// TwinCAT 3 PLC project SVLS_MOT
// ProgramVersion: 3.1.4026.15
// libraries:
//   LCLS General, * (SLAC)
//   lcls-twincat-math, * (SLAC - LCLS)
//   lcls-twincat-motion, * (SLAC)
//   PMPS, * (SLAC - LCLS)
//   Tc2_MC2, * (Beckhoff Automation GmbH)
//   Tc2_Standard, * (Beckhoff Automation GmbH)
//   Tc2_System, * (Beckhoff Automation GmbH)
//   Tc2_Utilities, * (Beckhoff Automation GmbH)
//   Tc3_Module, * (Beckhoff Automation GmbH)
//   TcUnit, * (www.tcunit.org)
// project tree:
//   DUTs/ ST_EPSLimits.TcDUT (not stored)
//   GVLs/ Main.TcGVL
//   ITFs/ I_ExternalSetpointGenerator.TcIO, I_HController.TcIO, I_CalculateHFromAngle.TcIO, I_MotionAxis.TcIO
//   / PlcTask.TcTTO, ProductionPlcTask.TcTTO, TestPlcTask.TcTTO
//   POUs/EPS/ FB_CheckEPS.TcPOU (not stored), FB_RestTimer.TcPOU (not stored), F_InRange.TcPOU (not stored), PRG_DET_Z_EPS.TcPOU
//   POUs/FBs/ FB_ExternalSetpointGenerator.TcPOU, FB_HController.TcPOU, FB_CalculateHFromAngle.TcPOU, FB_MotionAxisNC.TcPOU
//   POUs/ PRG_Main.TcPOU
//   Test/ FB_CalculateHFromAngle_Test.TcPOU, FB_HController_Test.TcPOU, FB_ExternalSetpointGenerator_Test.TcPOU, PRG_Test.TcPOU
// real-time tasks:
//   TASK PlcTask: cycle T#10ms, priority 20, ADS port 350
//   TASK TestPlcTask: cycle T#10ms, priority 1, ADS port 351
//   TASK ProductionPlcTask: cycle T#10ms, priority 2, ADS port 352
// motion (NC):
//   TASK SVLS_MOTION SAF: cycle T#2ms, priority 4, ADS port 501
//   TASK SVLS_MOTION SVB: cycle T#10ms, priority 8, ADS port 511
//   AXIS ExternalSetpointGenerator_Test2 (id 10)
//     OtherSettings: AllowMotionCmdToSlave=true, AllowMotionCmdToExtSetGenAxis=true
//     encoder EncType=1
//     drive DrvType=5
//       Analog: TorqueSetpointScale=10, ScaleFactorActTorque=0.1
//       TimeComp: TaskDelayCycles=1
//     controller CtrType=1
//       CtrPara: PriorControlFactor=1
//         Observer: BandWidth=20
//   AXIS ExternalSetpointGenerator_Test1 (id 9)
//     OtherSettings: AllowMotionCmdToSlave=true, AllowMotionCmdToExtSetGenAxis=true
//     encoder EncType=1
//     drive DrvType=5
//       Analog: TorqueSetpointScale=10, ScaleFactorActTorque=0.1
//       TimeComp: TaskDelayCycles=1
//     controller CtrType=1
//       CtrPara: PriorControlFactor=1
//         Observer: BandWidth=20
//   AXIS HControllerDetAngle_Test1 (id 11)
//     OtherSettings: AllowMotionCmdToSlave=true
//     encoder EncType=1
//     drive DrvType=5
//       Analog: TorqueSetpointScale=10, ScaleFactorActTorque=0.1
//       TimeComp: TaskDelayCycles=1
//     controller CtrType=1
//       CtrPara: PriorControlFactor=1
//         Observer: BandWidth=20
//   AXIS HControllerDetH_Test1 (id 12)
//     OtherSettings: AllowMotionCmdToSlave=true, AllowMotionCmdToExtSetGenAxis=true
//     encoder EncType=29
//       EncPara: ScaleFactorNumerator=1e-06, MaxCount=#xffffffff, MaxCountHighDWord=#x0000001f
//     drive DrvType=5
//       Analog: TorqueSetpointScale=10, ScaleFactorActTorque=0.1
//       TimeComp: TaskDelayCycles=1
//     controller CtrType=1
//       CtrPara: PriorControlFactor=1
//         PosDiffControl: Enable=false
//         Observer: BandWidth=20
//   AXIS M1_DET_Y_Angle (id 1)
//     General: UnitName=Degree
//     Dynamic: AccelerationMaximum=0.572958, DecelerationMaximum=0.572958, Acceleration=0.57, Deceleration=0.57
//     Velo: Maximum=0.02
//     OtherSettings: AllowMotionCmdToSlave=true
//     encoder EncType=29
//       EncPara: ScaleFactorNumerator=8.3819032e-08, Offset=-11223.9805, MaxCount=#xffffffff, MaxCountHighDWord=#x0000001f, ReferenceSystem=1
//         FilterTime: TVelo=0.1
//         Inc: RefSoftSyncMask=#x0000ffff
//     drive DrvType=24
//       Analog: VeloReferenz=0.025492, TorqueSetpointScale=10, ScaleFactorActTorque=0.1
//       TimeComp: TaskDelayCycles=1
//     controller CtrType=1
//       CtrPara: PriorControlFactor=1
//         PosDiffControl: Enable=false, Range=0.06
//         Observer: BandWidth=20
//   AXIS M2_DET_Z (id 2)
//     Dynamic: AccelerationMaximum=50, DecelerationMaximum=50, Acceleration=50, Deceleration=50
//     Velo: RefSearch=0.1, RefSync=0.1, SlowManual=0.25, FastManual=0.5, Maximum=0.5
//     TargetPosControl: Range=0.01
//     OtherSettings: AllowMotionCmdToSlave=true
//     encoder EncType=29
//       EncPara: ScaleFactorNumerator=5e-05, Offset=-6871872.3264, MaxCount=#xffffffff, MaxCountHighDWord=#x0000001f
//         SoftEndMinControl: Enable=true, Range=-53.8
//         SoftEndMaxControl: Enable=true, Range=51.3
//         Inc: RefSoftSyncMask=#x0000ffff
//     drive DrvType=24
//       Analog: VeloReferenz=0.5, TorqueSetpointScale=10, ScaleFactorActTorque=0.1
//       TimeComp: TaskDelayCycles=1
//     controller CtrType=1
//       CtrPara: PriorControlFactor=1
//         PosDiffControl: Range=0.07
//         Observer: BandWidth=20
//   AXIS M3_GRA_Y (id 3)
//     Dynamic: AccelerationMaximum=5, DecelerationMaximum=5, Acceleration=5, Deceleration=5, Jerk=5
//     Velo: RefSearch=0.01, RefSync=0.01, SlowManual=0.0025, FastManual=0.005, Maximum=0.05
//     PositionAreaControl: Range=0.003
//     TargetPosControl: Range=0.0002
//     OtherSettings: AllowMotionCmdToSlave=true
//     encoder EncType=29
//       EncPara: ScaleFactorNumerator=5e-05, Offset=-17.0296, MaxCount=#xffffffff, MaxCountHighDWord=#x0000001f
//         SoftEndMinControl: Enable=true, Range=-1.11
//         SoftEndMaxControl: Enable=true, Range=1.35
//         Inc: RefSoftSyncMask=#x0000ffff
//     drive DrvType=24
//       DrvPara: Inverse=true
//         Analog: VeloReferenz=0.106, TorqueSetpointScale=10, ScaleFactorActTorque=0.1
//         TimeComp: TaskDelayCycles=1
//     controller CtrType=1
//       CtrPara: PriorControlFactor=1
//         PosDiffControl: Range=0.1
//         Observer: BandWidth=20
//   AXIS M8_Det_Y_H (id 8)
//     Dynamic: AccelerationMaximum=100, DecelerationMaximum=100, Acceleration=1, Deceleration=1, Jerk=10
//     Velo: RefSearch=0.1, RefSync=0.1, SlowManual=0.25, FastManual=0.45, Maximum=0.25
//     PositionAreaControl: Enable=false, Range=1
//     TargetPosControl: Range=1, Time=1
//     OtherSettings: AllowMotionCmdToSlave=true, AllowMotionCmdToExtSetGenAxis=true, PulseDistancePos=1, PulseDistanceNeg=1
//     encoder EncType=29
//       EncPara: ScaleFactorNumerator=1e-06, MaxCount=#xffffffff, MaxCountHighDWord=#x0000001f
//         FilterTime: TVelo=1
//         SoftEndMinControl: Enable=true, Range=113
//         SoftEndMaxControl: Enable=true, Range=256
//         Inc: RefSoftSyncMask=#x0000ffff
//     drive DrvType=24
//       Analog: VeloReferenz=0.5, TorqueSetpointScale=10, ScaleFactorActTorque=0.1
//       TimeComp: TaskDelayCycles=1
//     controller CtrType=1
//       CtrPara: PriorControlFactor=1
//         PosDiffControl: Enable=false, Range=0.1
//         PID: PosKp=0
//         Observer: BandWidth=20
// I/O:
//   DEVICE Device 1 (EtherCAT), AmsNetId 199.4.42.250.2.1
//     EK1200_01_00 [EK1200-5000 EtherCAT Power supply (2A E-Bus)]
//       EL6070_01_00 [EL6070 1Ch. Licensing-Terminal]
//       EL7047_01_01-DET_Y [EL7047 1Ch. Stepper motor output stage (50V, 5A)]
//       EL5042_01_02-DET_Y-DET_Z [EL5042 2Ch. BiSS-C Encoder]
//       EL7047_01_03-DET_Z [EL7047 1Ch. Stepper motor output stage (50V, 5A)]
//       EL7047_01_04-GRT_Y [EL7047 1Ch. Stepper motor output stage (50V, 5A)]
//       EL5042_01_05-GRT_Y-SP5 [EL5042 2Ch. BiSS-C Encoder]
//       EL5042_01_06-SP1-SP2 [EL5042 2Ch. BiSS-C Encoder]
//       EL5042_01_07-SP3-SP4 [EL5042 2Ch. BiSS-C Encoder]
//       EL9011_01_Endstop [EL9011 End Terminal]
// variable links:
//   (this object) <-> Device 1 (EtherCAT)/EK1200_01_00/EL5042_01_02-DET_Y-DET_Z
//     Enc/Inputs/In/nComState @bit 1 <-> WcState/InputToggle
//     Enc/Inputs/In/nComState <-> WcState/WcState
//     Enc/Inputs/In/nDataIn1 <-> FB Inputs Channel 1/Position
//     Enc/Inputs/In/nDataIn1 <-> FB Inputs Channel 2/Position
//     Enc/Inputs/In/nState1 @bit 12 <-> FB Inputs Channel 1/Status/Diag
//     Enc/Inputs/In/nState1 @bit 12 <-> FB Inputs Channel 2/Status/Diag
//     Enc/Inputs/In/nState1 @bit 1 <-> FB Inputs Channel 1/Status/Error
//     Enc/Inputs/In/nState1 @bit 1 <-> FB Inputs Channel 2/Status/Error
//     Enc/Inputs/In/nState1 @bit 14 <-> FB Inputs Channel 1/Status/Input cycle counter
//     Enc/Inputs/In/nState1 @bit 14 <-> FB Inputs Channel 2/Status/Input cycle counter
//     Enc/Inputs/In/nState1 @bit 2 <-> FB Inputs Channel 1/Status/Ready
//     Enc/Inputs/In/nState1 @bit 2 <-> FB Inputs Channel 2/Status/Ready
//     Enc/Inputs/In/nState1 @bit 13 <-> FB Inputs Channel 1/Status/TxPDO State
//     Enc/Inputs/In/nState1 @bit 13 <-> FB Inputs Channel 2/Status/TxPDO State
//     Enc/Inputs/In/nState1 <-> FB Inputs Channel 1/Status/Warning
//     Enc/Inputs/In/nState1 <-> FB Inputs Channel 2/Status/Warning
//   (this object) <-> Device 1 (EtherCAT)/EK1200_01_00/EL7047_01_01-DET_Y
//     Drive/Inputs/In/nState1 @bit 3 <-> STM Status/Status/Error
//     Drive/Inputs/In/nState1 @bit 7 <-> STM Status/Status/Motor stall
//     Drive/Inputs/In/nState1 @bit 5 <-> STM Status/Status/Moving negative
//     Drive/Inputs/In/nState1 @bit 4 <-> STM Status/Status/Moving positive
//     Drive/Inputs/In/nState1 @bit 1 <-> STM Status/Status/Ready
//     Drive/Inputs/In/nState1 <-> STM Status/Status/Ready to enable
//     Drive/Inputs/In/nState1 @bit 6 <-> STM Status/Status/Torque reduced
//     Drive/Inputs/In/nState1 @bit 2 <-> STM Status/Status/Warning
//     Drive/Inputs/In/nState2 @bit 3 <-> STM Status/Status/Digital input 1
//     Drive/Inputs/In/nState2 @bit 4 <-> STM Status/Status/Digital input 2
//     Drive/Inputs/In/nState2 @bit 5 <-> STM Status/Status/Sync error
//     Drive/Inputs/In/nState2 @bit 7 <-> STM Status/Status/TxPDO Toggle
//     Drive/Inputs/In/nState4 @bit 1 <-> WcState/InputToggle
//     Drive/Inputs/In/nState4 <-> WcState/WcState
//     Drive/Outputs/Out/nCtrl1 <-> STM Control/Control/Enable
//     Drive/Outputs/Out/nCtrl1 @bit 2 <-> STM Control/Control/Reduce torque
//     Drive/Outputs/Out/nCtrl1 @bit 1 <-> STM Control/Control/Reset
//     Drive/Outputs/Out/nCtrl2 @bit 3 <-> STM Control/Control/Digital output 1
//     Drive/Outputs/Out/nDataOut2[0] <-> STM Velocity/Velocity
//   (this object) <-> Device 1 (EtherCAT)/EK1200_01_00/EL7047_01_03-DET_Z
//     Drive/Inputs/In/nState1 @bit 3 <-> STM Status/Status/Error
//     Drive/Inputs/In/nState1 @bit 7 <-> STM Status/Status/Motor stall
//     Drive/Inputs/In/nState1 @bit 5 <-> STM Status/Status/Moving negative
//     Drive/Inputs/In/nState1 @bit 4 <-> STM Status/Status/Moving positive
//     Drive/Inputs/In/nState1 @bit 1 <-> STM Status/Status/Ready
//     Drive/Inputs/In/nState1 <-> STM Status/Status/Ready to enable
//     Drive/Inputs/In/nState1 @bit 6 <-> STM Status/Status/Torque reduced
//     Drive/Inputs/In/nState1 @bit 2 <-> STM Status/Status/Warning
//     Drive/Inputs/In/nState2 @bit 3 <-> STM Status/Status/Digital input 1
//     Drive/Inputs/In/nState2 @bit 4 <-> STM Status/Status/Digital input 2
//     Drive/Inputs/In/nState2 @bit 5 <-> STM Status/Status/Sync error
//     Drive/Inputs/In/nState2 @bit 7 <-> STM Status/Status/TxPDO Toggle
//     Drive/Inputs/In/nState4 @bit 1 <-> WcState/InputToggle
//     Drive/Inputs/In/nState4 <-> WcState/WcState
//     Drive/Outputs/Out/nCtrl1 <-> STM Control/Control/Enable
//     Drive/Outputs/Out/nCtrl1 @bit 2 <-> STM Control/Control/Reduce torque
//     Drive/Outputs/Out/nCtrl1 @bit 1 <-> STM Control/Control/Reset
//     Drive/Outputs/Out/nCtrl2 @bit 3 <-> STM Control/Control/Digital output 1
//     Drive/Outputs/Out/nDataOut2[0] <-> STM Velocity/Velocity
//   (this object) <-> Device 1 (EtherCAT)/EK1200_01_00/EL5042_01_05-GRT_Y-SP5
//     Enc/Inputs/In/nComState @bit 1 <-> WcState/InputToggle
//     Enc/Inputs/In/nComState <-> WcState/WcState
//     Enc/Inputs/In/nDataIn1 <-> FB Inputs Channel 1/Position
//     Enc/Inputs/In/nState1 @bit 12 <-> FB Inputs Channel 1/Status/Diag
//     Enc/Inputs/In/nState1 @bit 1 <-> FB Inputs Channel 1/Status/Error
//     Enc/Inputs/In/nState1 @bit 14 <-> FB Inputs Channel 1/Status/Input cycle counter
//     Enc/Inputs/In/nState1 @bit 2 <-> FB Inputs Channel 1/Status/Ready
//     Enc/Inputs/In/nState1 @bit 13 <-> FB Inputs Channel 1/Status/TxPDO State
//     Enc/Inputs/In/nState1 <-> FB Inputs Channel 1/Status/Warning
//   (this object) <-> Device 1 (EtherCAT)/EK1200_01_00/EL7047_01_04-GRT_Y
//     Drive/Inputs/In/nState1 @bit 3 <-> STM Status/Status/Error
//     Drive/Inputs/In/nState1 @bit 7 <-> STM Status/Status/Motor stall
//     Drive/Inputs/In/nState1 @bit 5 <-> STM Status/Status/Moving negative
//     Drive/Inputs/In/nState1 @bit 4 <-> STM Status/Status/Moving positive
//     Drive/Inputs/In/nState1 @bit 1 <-> STM Status/Status/Ready
//     Drive/Inputs/In/nState1 <-> STM Status/Status/Ready to enable
//     Drive/Inputs/In/nState1 @bit 6 <-> STM Status/Status/Torque reduced
//     Drive/Inputs/In/nState1 @bit 2 <-> STM Status/Status/Warning
//     Drive/Inputs/In/nState2 @bit 3 <-> STM Status/Status/Digital input 1
//     Drive/Inputs/In/nState2 @bit 4 <-> STM Status/Status/Digital input 2
//     Drive/Inputs/In/nState2 @bit 5 <-> STM Status/Status/Sync error
//     Drive/Inputs/In/nState2 @bit 7 <-> STM Status/Status/TxPDO Toggle
//     Drive/Inputs/In/nState4 @bit 1 <-> WcState/InputToggle
//     Drive/Inputs/In/nState4 <-> WcState/WcState
//     Drive/Outputs/Out/nCtrl1 <-> STM Control/Control/Enable
//     Drive/Outputs/Out/nCtrl1 @bit 2 <-> STM Control/Control/Reduce torque
//     Drive/Outputs/Out/nCtrl1 @bit 1 <-> STM Control/Control/Reset
//     Drive/Outputs/Out/nCtrl2 @bit 3 <-> STM Control/Control/Digital output 1
//     Drive/Outputs/Out/nDataOut2[0] <-> STM Velocity/Velocity
//   SVLS_MOT Instance <-> Device 1 (EtherCAT)/EK1200_01_00/EL5042_01_02-DET_Y-DET_Z
//     ProductionPlcTask Inputs/Main.M1.nRawEncoderULINT <-> FB Inputs Channel 1/Position
//     ProductionPlcTask Inputs/Main.M2.nRawEncoderULINT <-> FB Inputs Channel 2/Position
//   SVLS_MOT Instance <-> Device 1 (EtherCAT)/EK1200_01_00/EL5042_01_05-GRT_Y-SP5
//     ProductionPlcTask Inputs/Main.M3.nRawEncoderULINT <-> FB Inputs Channel 1/Position
//   SVLS_MOT Instance <-> Device 1 (EtherCAT)/EK1200_01_00/EL7047_01_01-DET_Y
//     ProductionPlcTask Inputs/Main.M1.bLimitBackwardEnable <-> STM Status/Status/Digital input 2
//     ProductionPlcTask Inputs/Main.M8.bLimitBackwardEnable <-> STM Status/Status/Digital input 2
//     ProductionPlcTask Inputs/Main.M1.bLimitForwardEnable <-> STM Status/Status/Digital input 1
//     ProductionPlcTask Inputs/Main.M8.bLimitForwardEnable <-> STM Status/Status/Digital input 1
//   SVLS_MOT Instance <-> Device 1 (EtherCAT)/EK1200_01_00/EL7047_01_03-DET_Z
//     ProductionPlcTask Inputs/Main.M2.bLimitBackwardEnable <-> STM Status/Status/Digital input 2
//     ProductionPlcTask Inputs/Main.M2.bLimitForwardEnable <-> STM Status/Status/Digital input 1
//   SVLS_MOT Instance <-> Device 1 (EtherCAT)/EK1200_01_00/EL7047_01_04-GRT_Y
//     ProductionPlcTask Inputs/Main.M3.bLimitBackwardEnable <-> STM Status/Status/Digital input 2
//     ProductionPlcTask Inputs/Main.M3.bLimitForwardEnable <-> STM Status/Status/Digital input 1
//   SVLS_MOT Instance <-> SVLS_MOTION SAF/Axes/ExternalSetpointGenerator_Test1
//     TestPlcTask Inputs/PRG_Test.AxisReference_ExternalSetpointGenerator_Test1.NcToPlc <-> Outputs/ToPlc
//     TestPlcTask Outputs/PRG_Test.AxisReference_ExternalSetpointGenerator_Test1.PlcToNc <-> Inputs/FromPlc
//   SVLS_MOT Instance <-> SVLS_MOTION SAF/Axes/ExternalSetpointGenerator_Test2
//     TestPlcTask Inputs/PRG_Test.AxisReference_ExternalSetpointGenerator_Test2.NcToPlc <-> Outputs/ToPlc
//     TestPlcTask Outputs/PRG_Test.AxisReference_ExternalSetpointGenerator_Test2.PlcToNc <-> Inputs/FromPlc
//   SVLS_MOT Instance <-> SVLS_MOTION SAF/Axes/HControllerDetAngle_Test1
//     TestPlcTask Inputs/PRG_Test.stMotionStage_HControllerDetAngle_Test1.Axis.NcToPlc <-> Outputs/ToPlc
//     TestPlcTask Outputs/PRG_Test.stMotionStage_HControllerDetAngle_Test1.Axis.PlcToNc <-> Inputs/FromPlc
//   SVLS_MOT Instance <-> SVLS_MOTION SAF/Axes/HControllerDetH_Test1
//     PlcTask Outputs/PRG_Test.fbHController_Test.nDetAngleEncoderComState_Test1 <-> Enc/Inputs/In/nComState
//     PlcTask Outputs/PRG_Test.fbHController_Test.nDetAngleEncoderState1_Test1 <-> Enc/Inputs/In/nState1
//     TestPlcTask Inputs/PRG_Test.stMotionStage_HControllerDetH_Test1.Axis.NcToPlc <-> Outputs/ToPlc
//     TestPlcTask Outputs/PRG_Test.stMotionStage_HControllerDetH_Test1.Axis.PlcToNc <-> Inputs/FromPlc
//   SVLS_MOT Instance <-> SVLS_MOTION SAF/Axes/M1_DET_Y_Angle
//     ProductionPlcTask Inputs/Main.M1.Axis.NcToPlc <-> Outputs/ToPlc
//     ProductionPlcTask Outputs/Main.M1.Axis.PlcToNc <-> Inputs/FromPlc
//   SVLS_MOT Instance <-> SVLS_MOTION SAF/Axes/M2_DET_Z
//     ProductionPlcTask Inputs/Main.M2.Axis.NcToPlc <-> Outputs/ToPlc
//     ProductionPlcTask Outputs/Main.M2.Axis.PlcToNc <-> Inputs/FromPlc
//   SVLS_MOT Instance <-> SVLS_MOTION SAF/Axes/M3_GRA_Y
//     ProductionPlcTask Inputs/Main.M3.Axis.NcToPlc <-> Outputs/ToPlc
//     ProductionPlcTask Outputs/Main.M3.Axis.PlcToNc <-> Inputs/FromPlc
//   SVLS_MOT Instance <-> SVLS_MOTION SAF/Axes/M8_Det_Y_H
//     ProductionPlcTask Inputs/Main.M8.Axis.NcToPlc <-> Outputs/ToPlc
//     ProductionPlcTask Outputs/Main.M8.Axis.PlcToNc <-> Inputs/FromPlc
//     ProductionPlcTask Outputs/PRG_Main.fbHController.nEncoderCounts <-> Enc/Inputs/In/nDataIn1
//   SVLS_MOT Instance <-> SVLS_MOT/SVLS_MOT Instance
//     ProductionPlcTask Inputs/Main.M8.nRawEncoderULINT <-> ProductionPlcTask Outputs/PRG_Main.fbHController.nEncoderCounts
//     ProductionPlcTask Outputs/PRG_Main.fbHController.nEncoderCounts <-> ProductionPlcTask Inputs/Main.M8.nRawEncoderULINT

CONFIGURATION SVLS_MOT
    RESOURCE PLC ON TwinCAT3
        TASK PlcTask(INTERVAL := T#10ms, PRIORITY := 20);
        TASK ProductionPlcTask(INTERVAL := T#10ms, PRIORITY := 2);
        TASK TestPlcTask(INTERVAL := T#10ms, PRIORITY := 1);
        PROGRAM PRG_Main WITH ProductionPlcTask : PRG_Main;
        PROGRAM PRG_Test WITH TestPlcTask : PRG_Test;
    END_RESOURCE
END_CONFIGURATION

// ---- GVLs/Main.TcGVL

{attribute 'qualified_only'}
VAR_GLOBAL
    {attribute 'pytmc' := 'pv: CRIXS:SVLS:DET:MMS:Y_Angle'}
    {attribute 'TcLinkTo' := '.bLimitForwardEnable  := TIIB[EL7047_01_01-DET_Y]^STM Status^Status^Digital input 1;
                              .bLimitBackwardEnable := TIIB[EL7047_01_01-DET_Y]^STM Status^Status^Digital input 2;
                              .nRawEncoderULINT     := TIIB[EL5042_01_02-DET_Y-DET_Z]^FB Inputs Channel 1^Position'}
    M1: ST_MotionStage := (sName := 'CRIXS:SVLS:DET:MMS:Y_Angle');

    {attribute 'pytmc' := 'pv: CRIXS:SVLS:DET:MMS:Z'}
    {attribute 'TcLinkTo' := '.bLimitForwardEnable  := TIIB[EL7047_01_03-DET_Z]^STM Status^Status^Digital input 1;
                              .bLimitBackwardEnable := TIIB[EL7047_01_03-DET_Z]^STM Status^Status^Digital input 2;
                              .nRawEncoderULINT     := TIIB[EL5042_01_02-DET_Y-DET_Z]^FB Inputs Channel 2^Position'}
    M2: ST_MotionStage := (sName := 'CRIXS:SVLS:DET:MMS:Z');

    {attribute 'pytmc' := 'pv: CRIXS:SVLS:GRA:MMS:Y'}
    {attribute 'TcLinkTo' := '.bLimitForwardEnable  := TIIB[EL7047_01_04-GRT_Y]^STM Status^Status^Digital input 1;
                              .bLimitBackwardEnable := TIIB[EL7047_01_04-GRT_Y]^STM Status^Status^Digital input 2;
                              .nRawEncoderULINT     := TIIB[EL5042_01_05-GRT_Y-SP5]^FB Inputs Channel 1^Position'}
    M3: ST_MotionStage := (sName := 'CRIXS:SVLS:GRA:MMS:Y');

    {attribute 'pytmc' := 'pv:	CRIXS:SVLS:DET:MMS:Y_H'}
    {attribute 'TcLinkTo' := '.bLimitForwardEnable  := TIIB[EL7047_01_01-DET_Y]^STM Status^Status^Digital input 1;
                              .bLimitBackwardEnable := TIIB[EL7047_01_01-DET_Y]^STM Status^Status^Digital input 2;
                              .nRawEncoderULINT     := TIPC^SVLS_MOT^SVLS_MOT Instance^ProductionPlcTask Outputs^PRG_Main.fbHController.nEncoderCounts'}
    M8 : ST_MotionStage := (sName := 'CRIXS:SVLS:DET:MMS:Y_H');
	
END_VAR

// ---- ITFs/I_ExternalSetpointGenerator.TcIO
INTERFACE I_ExternalSetpointGenerator


METHOD Disable
VAR_OUTPUT
    Done : BOOL;
    Busy : BOOL;
    Error : BOOL;
    ErrorID : UDINT;
    Enabled : BOOL;
END_VAR
END_METHOD

PROPERTY DisableBusy : BOOL
GET
END_GET
END_PROPERTY

PROPERTY DisableDone : BOOL
GET
END_GET
END_PROPERTY


METHOD Enable
VAR_OUTPUT
    Done : BOOL;
    Busy : BOOL;
    Error : BOOL;
    ErrorID : UDINT;
    Enabled : BOOL;
END_VAR
END_METHOD

PROPERTY EnableBusy : BOOL
GET
END_GET
END_PROPERTY

PROPERTY EnableDone : BOOL
GET
END_GET
END_PROPERTY

PROPERTY EnableError : BOOL
GET
END_GET
END_PROPERTY


METHOD Halt
VAR_OUTPUT
    Done : BOOL;
    Busy : BOOL;
    Active : BOOL;
    CommandAborted : BOOL;
    Error : BOOL;
    ErrorID : UDINT;
END_VAR
END_METHOD

PROPERTY HaltBusy : BOOL
GET
END_GET
END_PROPERTY

PROPERTY HaltDone : BOOL
GET
END_GET
END_PROPERTY


METHOD IsEnabled : BOOL
END_METHOD


METHOD SetAcceleraSetpoint
VAR_INPUT
    Setpoint : LREAL;
END_VAR
VAR_OUTPUT
	Error : BOOL;
	ErrorMsg : T_MaxString;
END_VAR
END_METHOD


METHOD SetPositionSetpoint
VAR_INPUT
    Setpoint : LREAL;
END_VAR
VAR_OUTPUT
	Error : BOOL;
	ErrorMsg : T_MaxString;
END_VAR
END_METHOD


METHOD SetSetpoints
VAR_INPUT
    PositionSetpoint : LREAL;
    VelocitySetpoint : LREAL;
    AcceleraSetpoint : LREAL;
END_VAR
VAR_OUTPUT
	Error : BOOL;
	ErrorMsg : T_MaxString;
END_VAR
END_METHOD


METHOD SetVelocitySetpoint
VAR_INPUT
    Setpoint : LREAL;
END_VAR
VAR_OUTPUT
	Error : BOOL;
	ErrorMsg : T_MaxString;
END_VAR
END_METHOD

END_INTERFACE

// ---- ITFs/I_HController.TcIO
INTERFACE I_HController

END_INTERFACE

// ---- ITFs/I_CalculateHFromAngle.TcIO
INTERFACE I_CalculateHFromAngle


METHOD CalculateH : LREAL
VAR_INPUT
    Radians : LREAL;
END_VAR
VAR_OUTPUT
    Error : BOOL;
    ErrorMsg : T_MaxString;
END_VAR
END_METHOD


METHOD CalculateHVelocity : LREAL
VAR_INPUT
    Radians : LREAL;
    RadiansPerSecond : LREAL;
END_VAR
VAR_OUTPUT
    Error : BOOL;
    ErrorMsg : T_MaxString;
END_VAR
END_METHOD

END_INTERFACE

// ---- ITFs/I_MotionAxis.TcIO

INTERFACE I_MotionAxis


METHOD GetAxisRef : REFERENCE TO AXIS_REF
END_METHOD


METHOD GetPowerOverride : LREAL
END_METHOD

PROPERTY MeasuredAcceleration : LREAL
GET
END_GET
END_PROPERTY

PROPERTY MeasuredPosition : LREAL
GET
END_GET
END_PROPERTY

PROPERTY MeasuredVelocity : LREAL
GET
END_GET
END_PROPERTY


METHOD MoveAbsolute
VAR_INPUT
    Position : LREAL; 
    Velocity : LREAL; 
    Acceleration : LREAL := 0.0; 
    Deceleration : LREAL := 0.0; 
    Jerk : LREAL := 0.0;
    BufferMode : MC_BufferMode := MC_BufferMode.MC_Aborting;
END_VAR
VAR_OUTPUT
    Done : BOOL;
    Busy : BOOL;
    Active : BOOL;
    CommandAborted : BOOL;
    Error : BOOL;
    ErrorID : UDINT;
    ErrorStr : T_MaxString;
END_VAR
END_METHOD

PROPERTY MoveAbsoluteBusy : BOOL
GET
END_GET
END_PROPERTY

PROPERTY MoveAbsoluteDone : BOOL
GET
END_GET
END_PROPERTY

PROPERTY MoveAbsoluteError : BOOL
GET
END_GET
END_PROPERTY

PROPERTY MoveAbsoluteErrorID : UDINT
GET
END_GET
END_PROPERTY

PROPERTY MoveAbsoluteTargetAcceleration : LREAL
GET
END_GET
END_PROPERTY

PROPERTY MoveAbsoluteTargetDeceleration : LREAL
GET
END_GET
END_PROPERTY

PROPERTY MoveAbsoluteTargetJerk : LREAL
GET
END_GET
END_PROPERTY

PROPERTY MoveAbsoluteTargetPosition : LREAL
GET
END_GET
END_PROPERTY

PROPERTY MoveAbsoluteTargetVelocity : LREAL
GET
END_GET
END_PROPERTY

PROPERTY NegativeMotionIsEnabled : BOOL
GET
END_GET
END_PROPERTY

PROPERTY PositiveMotionIsEnabled : BOOL
GET
END_GET
END_PROPERTY


METHOD Power
VAR_INPUT
    Enable : BOOL;
    Enable_Positive : BOOL;
    Enable_Negative : BOOL;
    Override : LREAL := 100.0; (* in percent from 0 to 100 *)
    BufferMode : MC_BufferMode := MC_BufferMode.MC_Aborting;
END_VAR
VAR_OUTPUT
    Status : BOOL;
    Busy : BOOL;
    Active : BOOL;
    Error : BOOL;
    ErrorID : UDINT;
    ErrorStr : T_MaxString;
END_VAR
END_METHOD

PROPERTY PowerError : BOOL
GET
END_GET
END_PROPERTY

PROPERTY PowerErrorID : UDINT
GET
END_GET
END_PROPERTY

PROPERTY PowerIsEnabled : BOOL
GET
END_GET
END_PROPERTY

PROPERTY PowerOverride : LREAL
GET
END_GET
END_PROPERTY

PROPERTY PowerStatus : BOOL
GET
END_GET
END_PROPERTY


METHOD Reset
VAR_OUTPUT
    Done    : BOOL;
    Busy    : BOOL;
    Error   : BOOL;
    ErrorID : UDINT;
    ErrorStr : T_MaxString;
END_VAR
END_METHOD


PROPERTY SetpointAcceleration : LREAL
GET
END_GET
END_PROPERTY


PROPERTY SetpointJerk : LREAL
GET
END_GET
END_PROPERTY


PROPERTY SetpointPosition : LREAL
GET
END_GET
END_PROPERTY


PROPERTY SetpointVelocity : LREAL
GET
END_GET
END_PROPERTY


METHOD SetPowerOverride
VAR_INPUT
    Override : LREAL; (* in percent from 0 to 100 *)
END_VAR
VAR_OUTPUT
    Status : BOOL;
    Busy : BOOL;
    Active : BOOL;
    Error : BOOL;
    ErrorID : UDINT;
    ErrorStr : T_MaxString;
END_VAR
END_METHOD

END_INTERFACE

// ---- POUs/PRG_Main.TcPOU

PROGRAM PRG_Main
VAR
    fbDetYAngle : FB_MotionStage;
    fbDetZ : FB_MotionStage;
    fbGraY : FB_MotionStage;
    fbDetYH : FB_MotionStage;
    bInit : BOOL := TRUE;

    fbMotionAxisDetAngle : FB_MotionAxisNC(
        AxisReference := Main.M1.Axis
    );
    fbMotionAxisDetH : FB_MotionAxisNC(
        AxisReference := Main.M8.Axis
    );
    fbCalculateHFromAngle : FB_CalculateHFromAngle(
        D_tu := 1238.29,
        R_a := 1200.10,
        R_c := 89.78
    );
    {attribute 'TcLinkTo' := '.nEncoderCount := TINC^SVLS_MOTION SAF^Axes^M8_Det_Y_H^Enc^Inputs^In^nDataIn1'}
    fbHController : FB_HController(
        iMotionAxisDetAngle := fbMotionAxisDetAngle,
        iCalculateHFromAngle := fbCalculateHFromAngle,
        stMotionStageAxisDetAngle := Main.M1,
        stMotionStageAxisDetH := Main.M8,
        bDetHMoveAbsoluteBusy := fbDetYH.fbDriveVirtual.fbMoveAbsolute.Busy
    );
	
END_VAR


IF bInit THEN
    bInit := FALSE;

    Main.M1.bHardwareEnable := TRUE;
    Main.M1.bPowerSelf := TRUE;
    Main.M1.nBrakeMode := ENUM_StageBrakeMode.NO_BRAKE;
    Main.M1.nEnableMode := ENUM_StageEnableMode.DURING_MOTION;

    Main.M2.bHardwareEnable := TRUE;
    Main.M2.bPowerSelf := TRUE;
    Main.M2.nBrakeMode := ENUM_StageBrakeMode.NO_BRAKE;
    Main.M2.nEnableMode := ENUM_StageEnableMode.DURING_MOTION;

    Main.M3.bHardwareEnable := TRUE;
    Main.M3.bPowerSelf := TRUE;
    Main.M3.nBrakeMode := ENUM_StageBrakeMode.NO_BRAKE;
    Main.M3.nEnableMode := ENUM_StageEnableMode.DURING_MOTION;

    Main.M8.bHardwareEnable := TRUE;
    Main.M8.bPowerSelf := TRUE;
    Main.M8.nBrakeMode := ENUM_StageBrakeMode.NO_BRAKE;
    Main.M8.nEnableMode := ENUM_StageEnableMode.DURING_MOTION;
END_IF

PRG_DET_Z_EPS();

fbDetYAngle(stMotionStage:=Main.M1);
fbHController();
fbDetYH(stMotionStage:=Main.M8);
fbDetZ(stMotionStage:=Main.M2);
fbGraY(stMotionStage:=Main.M3);

END_PROGRAM

// ---- POUs/FBs/FB_MotionAxisNC.TcPOU

FUNCTION_BLOCK FB_MotionAxisNC IMPLEMENTS I_MotionAxis
VAR CONSTANT
    nOFFSET_TO_PLCTONC_AXIS_REF_CTRL : DWORD := 0;
END_VAR
VAR
    AxisReference : REFERENCE TO AXIS_REF;

    AxisReference_PLCtoNC_ControlDWord : MC.PLCTONC_AXIS_REF_CTRL;

    fbMcReset : MC_Reset;
    bCommandedReset : BOOL;

    fbMcPower : MC_Power;

    bCommandedMoveAbsolute : BOOL;
    fbMcMoveAbsolute : MC_MoveAbsolute;

    bMostRecentMoveAbsoluteDone : BOOL;
END_VAR


AxisReference.ReadStatus();

MEMCPY(
    ADR(AxisReference_PLCtoNC_ControlDWord),
    ADR(AxisReference.PlcToNc) + nOFFSET_TO_PLCTONC_AXIS_REF_CTRL,
    SIZEOF(AxisReference_PLCtoNC_ControlDWord)
);

fbMcReset(
    Axis := AxisReference,
    Execute := bCommandedReset
);
bCommandedReset := FALSE;

fbMcPower(Axis := AxisReference);

// IF bCommandedMoveAbsolute THEN
// 	ADSLOGSTR(
// 		msgCtrlMask := ADSLOG_MSGTYPE_ERROR,
// 		msgFmtStr := 'Commanded move absolute.',
// 		strArg := ''
// 	);
// END_IF

fbMcMoveAbsolute(
    Axis := AxisReference,
    Execute := bCommandedMoveAbsolute
);
bCommandedMoveAbsolute := FALSE;

IF THIS^.fbMcMoveAbsolute.Done THEN
    THIS^.bMostRecentMoveAbsoluteDone := TRUE;
END_IF

//FB_Init is always available implicitly and it is used primarily for initialization.
//The return value is not evaluated. For a specific influence, you can also declare the
//methods explicitly and provide additional code there with the standard initialization
//code. You can evaluate the return value.
METHOD FB_Init: BOOL
VAR_INPUT
    bInitRetains: BOOL; // TRUE: the retain variables are initialized (reset warm / reset cold)
    bInCopyCode: BOOL;  // TRUE: the instance will be copied to the copy code afterward (online change)

    AxisReference : REFERENCE TO AXIS_REF;
END_VAR

THIS^.AxisReference REF= AxisReference;
END_METHOD


METHOD GetAxisRef : REFERENCE TO AXIS_REF

GetAxisRef REF= THIS^.AxisReference;
END_METHOD


METHOD GetPowerOverride : LREAL

GetPowerOverride := TO_LREAL(THIS^.AxisReference.PlcToNc.Override) / 10000.0;
END_METHOD


PROPERTY MeasuredAcceleration : LREAL
GET

MeasuredAcceleration := THIS^.AxisReference.NcToPlc.ActAcc;
END_GET
END_PROPERTY


PROPERTY MeasuredPosition : LREAL
GET

MeasuredPosition := THIS^.AxisReference.NcToPlc.ActPos;
END_GET
END_PROPERTY


PROPERTY MeasuredVelocity : LREAL
GET

MeasuredVelocity := THIS^.AxisReference.NcToPlc.ActVelo;
END_GET
END_PROPERTY


METHOD MoveAbsolute
VAR_INPUT
    Position	: LREAL;
    Velocity	: LREAL;
    Acceleration	: LREAL := 0.0;
    Deceleration	: LREAL := 0.0;
    Jerk	: LREAL := 0.0;
    BufferMode	: MC_BufferMode := MC_BufferMode.MC_Aborting;
END_VAR
VAR_OUTPUT
    Done	: BOOL;
    Busy	: BOOL;
    Active	: BOOL;
    CommandAborted	: BOOL;
    Error	: BOOL;
    ErrorID	: UDINT;
    ErrorStr	: T_MaxString;
END_VAR

IF NOT MoveAbsoluteBusy THEN
    bMostRecentMoveAbsoluteDone := FALSE;

    bCommandedMoveAbsolute := TRUE;
END_IF

THIS^.fbMcMoveAbsolute(
    Axis := THIS^.AxisReference,
    Position := Position,
    Velocity := Velocity,
    Acceleration := Acceleration,
    Deceleration := Deceleration,
    Jerk := Jerk,
    BufferMode := BufferMode,
    Done => Done,
    Busy => Busy,
    Active => Active,
    CommandAborted => CommandAborted,
    Error => Error,
    ErrorID => ErrorID
);

ErrorStr := '';
END_METHOD


PROPERTY MoveAbsoluteBusy : BOOL
GET

MoveAbsoluteBusy := THIS^.fbMcMoveAbsolute.Busy;
END_GET
END_PROPERTY


PROPERTY MoveAbsoluteDone : BOOL
GET

MoveAbsoluteDone := THIS^.fbMcMoveAbsolute.Done OR THIS^.bMostRecentMoveAbsoluteDone;
END_GET
END_PROPERTY


PROPERTY MoveAbsoluteError : BOOL
GET

MoveAbsoluteError := THIS^.fbMcMoveAbsolute.Error;
END_GET
END_PROPERTY


PROPERTY MoveAbsoluteErrorID : UDINT
GET

MoveAbsoluteErrorID := THIS^.fbMcMoveAbsolute.ErrorID;
END_GET
END_PROPERTY


PROPERTY MoveAbsoluteTargetAcceleration : LREAL
GET

MoveAbsoluteTargetAcceleration := THIS^.fbMcMoveAbsolute.Acceleration;
END_GET
END_PROPERTY


PROPERTY MoveAbsoluteTargetDeceleration : LREAL
GET

MoveAbsoluteTargetDeceleration := THIS^.fbMcMoveAbsolute.Deceleration;
END_GET
END_PROPERTY


PROPERTY MoveAbsoluteTargetJerk : LREAL
GET

MoveAbsoluteTargetJerk := THIS^.fbMcMoveAbsolute.Jerk;
END_GET
END_PROPERTY


PROPERTY MoveAbsoluteTargetPosition : LREAL
GET

MoveAbsoluteTargetPosition := THIS^.fbMcMoveAbsolute.Position;
END_GET
END_PROPERTY


PROPERTY MoveAbsoluteTargetVelocity : LREAL
GET

MoveAbsoluteTargetVelocity := THIS^.fbMcMoveAbsolute.Velocity;
END_GET
END_PROPERTY


PROPERTY NegativeMotionIsEnabled : BOOL
GET

NegativeMotionIsEnabled := THIS^.AxisReference_PLCtoNC_ControlDWord.2;;
END_GET
END_PROPERTY


PROPERTY PositiveMotionIsEnabled : BOOL
GET

PositiveMotionIsEnabled := THIS^.AxisReference_PLCtoNC_ControlDWord.1;
END_GET
END_PROPERTY


METHOD Power
VAR_INPUT
    Enable	: BOOL;
    Enable_Positive	: BOOL;
    Enable_Negative	: BOOL;
    (* in percent from 0 to 100 *)
    Override	: LREAL := 100.0;
    BufferMode	: MC_BufferMode := MC_BufferMode.MC_Aborting;
END_VAR
VAR_OUTPUT
    Status	: BOOL;
    Busy	: BOOL;
    Active	: BOOL;
    Error	: BOOL;
    ErrorID	: UDINT;
    ErrorStr	: T_MaxString;
END_VAR

THIS^.fbMcPower(
    Axis := THIS^.AxisReference,
    Enable := Enable,
    Enable_Positive := Enable_Positive,
    Enable_Negative := Enable_Negative,
    Override := Override,
    BufferMode := BufferMode,
    Status => Status,
    Busy => Busy,
    Active => Active,
    Error => Error,
    ErrorID => ErrorID
);

ErrorStr := '';
END_METHOD


PROPERTY PowerError : BOOL
GET

PowerError := THIS^.fbMcPower.Error;
END_GET
END_PROPERTY


PROPERTY PowerErrorID : UDINT
GET

PowerErrorID := THIS^.fbMcPower.ErrorID;
END_GET
END_PROPERTY


METHOD PowerErrorIDToStr : T_MaxString
VAR_INPUT
    ErrorID : UDINT;
END_VAR

PowerErrorIDToStr := '';
END_METHOD


PROPERTY PowerIsEnabled : BOOL
GET

PowerIsEnabled := THIS^.AxisReference_PLCtoNC_ControlDWord.0;
END_GET
END_PROPERTY


PROPERTY PowerOverride : LREAL
GET

PowerOverride := GetPowerOverride();
END_GET
END_PROPERTY


PROPERTY PowerStatus : BOOL
GET

PowerStatus := THIS^.fbMcPower.Status;
END_GET
END_PROPERTY


METHOD Reset
VAR_OUTPUT
    Done : BOOL;
    Busy : BOOL;
    Error : BOOL;
    ErrorID : UDINT;
    ErrorStr : T_MaxString;
END_VAR

bCommandedReset := TRUE;

THIS^.fbMcReset(
    Axis := THIS^.AxisReference,
    Done => Done,
    Busy => Busy,
    Error => Error,
    ErrorID => ErrorID,
);

ErrorStr := '';
END_METHOD


PROPERTY SetpointAcceleration : LREAL
GET

SetpointAcceleration := THIS^.AxisReference.NcToPlc.SetAcc;
END_GET
END_PROPERTY


PROPERTY SetpointJerk : LREAL
GET

SetpointJerk := THIS^.AxisReference.NcToPlc.SetJerk;
END_GET
END_PROPERTY


PROPERTY SetpointPosition : LREAL
GET

SetpointPosition := THIS^.AxisReference.NcToPlc.SetPos;
END_GET
END_PROPERTY


PROPERTY SetpointVelocity : LREAL
GET

SetpointVelocity := THIS^.AxisReference.NcToPlc.SetVelo;
END_GET
END_PROPERTY


METHOD SetPowerOverride
VAR_INPUT
    (* in percent from 0 to 100 *)
    Override	: LREAL;
END_VAR
VAR_OUTPUT
    Status	: BOOL;
    Busy	: BOOL;
    Active	: BOOL;
    Error	: BOOL;
    ErrorID	: UDINT;
    ErrorStr	: T_MaxString;
END_VAR

THIS^.fbMcPower(
    Axis := THIS^.AxisReference,
    Override := Override,
    Status => Status,
    Busy => Busy,
    Error => Error,
    ErrorID => ErrorID
);

ErrorStr := '';
END_METHOD

END_FUNCTION_BLOCK

// ---- POUs/FBs/FB_CalculateHFromAngle.TcPOU

{attribute 'no_explicit_call' := 'Do not call this POU directly'}
FUNCTION_BLOCK FB_CalculateHFromAngle IMPLEMENTS I_CalculateHFromAngle
VAR
    D_tu : LREAL;
    R_c : LREAL;
    R_a : LREAL;
END_VAR


METHOD PUBLIC CalculateH : LREAL
VAR_INPUT
    Radians : LREAL;
END_VAR
VAR_OUTPUT
    Error : BOOL;
    ErrorMsg : T_MaxString;
END_VAR
VAR
    a : LREAL;
    b : LREAL;
    c : LREAL;
    d : LREAL;
    e : LREAL;
    f : LREAL;
    g : LREAL;
    h : LREAL;
    //sqrt_operand : LREAL;
END_VAR

IF R_c = 0 THEN
    Error := TRUE;
    ErrorMsg := CONCAT('R_c cannot equal 0. Value: ', TO_STRING(R_c));
    RETURN;
END_IF

a := R_a * COS(Radians);
b := D_tu - a;
c := b / R_c;

IF c < -1.0 OR c > 1.0 THEN
    Error := TRUE;
    ErrorMsg := CONCAT('Invalid angle. Value: ', TO_STRING(Radians));
    RETURN;
END_IF

d := ACOS(c);
e := SIN(d);
f := SIN(Radians);
g := R_a * f;
h := R_c * e;

CalculateH := h + g;

(*
sqrt_operand := -EXPT(R_a,2) * EXPT(COS(Angle),2) + 2 * R_a * D_tu * COS(Angle) + R_c - EXPT(D_tu,2);

IF sqrt_operand < 0.0 THEN
    Error := TRUE;
    ErrorMsg := CONCAT('Invalid angle. Value: ', TO_STRING(Angle));
    RETURN;
END_IF

CalculateH := R_a * SIN(Angle) - SQRT(sqrt_operand);
*)
END_METHOD


METHOD CalculateHVelocity : LREAL
VAR_INPUT
    Radians : LREAL;
    RadiansPerSecond : LREAL;
END_VAR
VAR_OUTPUT
    Error : BOOL;
    ErrorMsg : T_MaxString;
END_VAR
VAR
    A : LREAL;
    b : LREAL;
    b_dot : LREAL;
    C : LREAL;
    D : LREAL;
    fNumberToSqrt : LREAL;
END_VAR

A := R_a;
b := Radians;
b_dot := RadiansPerSecond;
C := R_c;
D := D_tu;
fNumberToSqrt := 1 - EXPT((D - (A * COS(b))/C), 2);

IF fNumberToSqrt <= 0 THEN
    Error := TRUE;
    ErrorMsg := 'number to sqrt was 0 or less than 0.';
    RETURN;
END_IF

CalculateHVelocity := A * b_dot * (COS(b) - (SIN(b)*(D - (COS(b))/C))/(SQRT(fNumberToSqrt)));
END_METHOD


METHOD FB_Init: BOOL
VAR_INPUT
    bInitRetains: BOOL; // TRUE: the retain variables are initialized (reset warm / reset cold)
    bInCopyCode: BOOL;  // TRUE: the instance will be copied to the copy code afterward (online change)

    D_tu : LREAL;
    R_c : LREAL;
    R_a : LREAL;
END_VAR

THIS^.D_tu := D_tu;
THIS^.R_c := R_c;
THIS^.R_a := R_a;
END_METHOD

END_FUNCTION_BLOCK

// ---- POUs/FBs/FB_HController.TcPOU

FUNCTION_BLOCK FB_HController IMPLEMENTS I_HController
VAR
    iMotionAxisDetAngle : I_MotionAxis;
    iCalculateHFromAngle : I_CalculateHFromAngle;
    stMotionStageAxisDetAngle : REFERENCE TO ST_MotionStage;
    stMotionStageAxisDetH : REFERENCE TO ST_MotionStage;
    bDetHMoveAbsoluteBusy : REFERENCE TO BOOL;

    fHPositionMeasured : LREAL;
    fHPositionSetpoint : LREAL;

    fHPositionGain : LREAL;
    fHPositionAdjustmentIntegration : LREAL;

    nEncoderCounts AT %Q* : ULINT; // nm/count

    rtMoveCmdTrigger : R_TRIG;
    ftResetTrigger : F_TRIG;
END_VAR


fHPositionMeasured := iCalculateHFromAngle.CalculateH(
    Radians := DEG_TO_RAD(iMotionAxisDetAngle.MeasuredPosition)
);

nEncoderCounts := TO_ULINT(fHPositionMeasured * 1E6);

fHPositionSetpoint := iCalculateHFromAngle.CalculateH(
    Radians := DEG_TO_RAD(iMotionAxisDetAngle.SetpointPosition)
);

rtMoveCmdTrigger(CLK := stMotionStageAxisDetAngle.bExecute);

IF rtMoveCmdTrigger.Q THEN
    stMotionStageAxisDetH.bMoveCmd := TRUE;
    stMotionStageAxisDetH.fPosition := iCalculateHFromAngle.CalculateH(
        Radians := DEG_TO_RAD(stMotionStageAxisDetAngle.fPosition)
    );
    stMotionStageAxisDetH.fVelocity := stMotionStageAxisDetH.stAxisParameters.fVeloMaximum *
        stMotionStageAxisDetAngle.fVelocity / stMotionStageAxisDetAngle.stAxisParameters.fVeloMaximum;
END_IF

ftResetTrigger(CLK := bDetHMoveAbsoluteBusy);

IF ftResetTrigger.Q THEN
    stMotionStageAxisDetAngle.bReset := TRUE;
    stMotionStageAxisDetH.bReset := TRUE;
END_IF


METHOD FB_Init: BOOL
VAR_INPUT
    bInitRetains: BOOL; // TRUE: the retain variables are initialized (reset warm / reset cold)
    bInCopyCode: BOOL;  // TRUE: the instance will be copied to the copy code afterward (online change)

    iMotionAxisDetAngle : I_MotionAxis;
    iCalculateHFromAngle : I_CalculateHFromAngle;
    stMotionStageAxisDetAngle : REFERENCE TO ST_MotionStage;
    stMotionStageAxisDetH : REFERENCE TO ST_MotionStage;
    bDetHMoveAbsoluteBusy : REFERENCE TO BOOL;

END_VAR

THIS^.iMotionAxisDetAngle := iMotionAxisDetAngle;
THIS^.iCalculateHFromAngle := iCalculateHFromAngle;
THIS^.stMotionStageAxisDetAngle REF= stMotionStageAxisDetAngle;
THIS^.stMotionStageAxisDetH REF= stMotionStageAxisDetH;
THIS^.bDetHMoveAbsoluteBusy REF= bDetHMoveAbsoluteBusy;
END_METHOD

END_FUNCTION_BLOCK

// ---- POUs/EPS/PRG_DET_Z_EPS.TcPOU
PROGRAM PRG_DET_Z_EPS
VAR
	{attribute 'pytmc' := 'pv: SVLS:DET:MMS:Z:EPS'}
    aDET_Z_EPS		: ARRAY [1 .. 2] OF ST_EPSLimits;
	
    {attribute 'pytmc' := 'pv: CRIX:DPL:MMS:X:EPS:OVRD_MODE'}
    bEPS_Override : BOOL := FALSE;
    {attribute 'pytmc' := 'pv: CRIX:DPL:MMS:X:EPS:OVRD_COUNTDOWN'}
    tEPS_TimerCountDown : STRING := TIME_TO_STRING(T#0S);
	tEPS_OVRD_RESET_TIME : TIME := T#5M;
    fbResetTimer : FB_RestTimer;
	
	
	bInit : BOOL := TRUE;
	
	fDET_Z : LREAL;
	fDET_Y_ANGLE : LREAL ;
	fDET_Y_ANGLE_VALUE : LREAL := 6;
	bYAngleBelow : BOOL;

    fbEPS : FB_EPS;
    fbCheckEPS : FB_CheckEPS;
END_VAR

fDET_Y_ANGLE := Main.M1.stAxisStatus.fActPosition;
fDET_Z := Main.M2.stAxisStatus.fActPosition;

IF bInit THEN
    // Set Inital Values
    aDET_Z_EPS[1].fBwd_Limits := -53.8;
    aDET_Z_EPS[1].fFwd_Limits := 35;
	
    aDET_Z_EPS[2].fBwd_Limits := -45;
    aDET_Z_EPS[2].fFwd_Limits := 51.3;

    bInit := FALSE;
END_IF

IF fDET_Y_ANGLE > fDET_Y_ANGLE_VALUE THEN bYAngleBelow := FALSE; ELSE bYAngleBelow := TRUE; END_IF
	
fbEPS(eps:=aDET_Z_EPS[1].stEPS);
fbEPS.setMessage('DET_Y_ANGLE < 6');
fbEPS.setBit(0, bYAngleBelow);

fbEPS(eps:=aDET_Z_EPS[2].stEPS);
fbEPS.setMessage('DET_Y_ANGLE > 6');
fbEPS.setBit(0, NOT bYAngleBelow);


fbResetTimer(bInput:=bEPS_Override, tElapseTime:=tEPS_OVRD_RESET_TIME, tCountDown:=tEPS_TimerCountDown);
fbCheckEPS(stMotor:= Main.M2, fPosition:=fDET_Z, aEPSLimits:= aDET_Z_EPS, stForwardMotorEPS:=Main.M2.stEPSForwardEnable, stBackwardMotorEPS:= Main.M2.stEPSBackwardEnable, bEPS_Override:=bEPS_Override);

END_PROGRAM

// ---- Test/PRG_Test.TcPOU

PROGRAM PRG_Test
VAR
    fbCalculateHFromAngle_Test : FB_CalculateHFromAngle_Test;

    AxisReference_ExternalSetpointGenerator_Test1 : AXIS_REF;
    MotionAxis_ExternalSetpointGenerator_Test1 : FB_MotionAxisNC(
        AxisReference := AxisReference_ExternalSetpointGenerator_Test1
    );
    AxisReference_ExternalSetpointGenerator_Test2 : AXIS_REF;
    MotionAxis_ExternalSetpointGenerator_Test2 : FB_MotionAxisNC(
        AxisReference := AxisReference_ExternalSetpointGenerator_Test2
    );
    fbExternalSetpointGenerator_Test : FB_ExternalSetpointGenerator_Test(
        MotionAxis_Test1 := MotionAxis_ExternalSetpointGenerator_Test1,
        MotionAxis_Test2 := MotionAxis_ExternalSetpointGenerator_Test2
    );

    stMotionStage_HControllerDetAngle_Test1 : ST_MotionStage;
    stMotionStage_HControllerDetH_Test1 : ST_MotionStage;

    //AxisReference_HControllerDetAngle_Test1 : AXIS_REF;
    MotionAxis_HControllerDetAngle_Test1 : FB_MotionAxisNC(
        AxisReference := stMotionStage_HControllerDetAngle_Test1.Axis
    );
    //AxisReference_HControllerDetH_Test1 : AXIS_REF;
    MotionAxis_HControllerDetH_Test1 : FB_MotionAxisNC(
        AxisReference := stMotionStage_HControllerDetH_Test1.Axis
    );
    fbHController_Test : FB_HController_Test(
        MotionAxisDetAngle_Test1 := MotionAxis_HControllerDetAngle_Test1,
        MotionAxisDetH_Test1 := MotionAxis_HControllerDetH_Test1
    );
    fbMotionStage_HControllerDetAngle_Test1 : FB_MotionStage;
    fbMotionStage_HControllerDetH_Test1 : FB_MotionStage;
END_VAR


MotionAxis_ExternalSetpointGenerator_Test1();
MotionAxis_ExternalSetpointGenerator_Test2();
MotionAxis_HControllerDetAngle_Test1();
MotionAxis_HControllerDetH_Test1();

fbMotionStage_HControllerDetAngle_Test1(stMotionStage := stMotionStage_HControllerDetAngle_Test1);
fbMotionStage_HControllerDetH_Test1(stMotionStage := stMotionStage_HControllerDetH_Test1);

TcUnit.RUN();

END_PROGRAM

// ---- Test/FB_CalculateHFromAngle_Test.TcPOU

FUNCTION_BLOCK FB_CalculateHFromAngle_Test EXTENDS FB_TestSuite


TestCalculateHExpectCorrectValue();


METHOD PRIVATE TestCalculateHExpectCorrectValue
VAR
    fAngleDegrees : LREAL;
    fAngleRadians : LREAL;
    fExpected : LREAL;
    fAllowableDelta : LREAL := 1e-3;

    fbCalculateHFromAngle : FB_CalculateHFromAngle(
        D_tu := 1239.5,
        R_a := 1200,
        R_c := 90
    );
    fResult : LREAL;
END_VAR

(*

Precomputed expected values. Using subset for tests.

length_1	angle_1	length_2	angle_2	length_3	angle_3	length_4	angle_4
258.8987	270	    90	        53	    1200	    8.9662	1.2395e+03	180
258.1957	270	    90	        53.1000	1200	    8.9276	1.2395e+03	180
257.4880	270	    90	        53.2000	1200	    8.8889	1.2395e+03	180
256.7754	270	    90	        53.3000	1200	    8.8499	1.2395e+03	180
256.0580	270	    90	        53.4000	1200	    8.8107	1.2395e+03	180
255.3356	270	    90	        53.5000	1200	    8.7713	1.2395e+03	180
254.6081	270	    90	        53.6000	1200	    8.7316	1.2395e+03	180
253.8756	270	    90	        53.7000	1200	    8.6917	1.2395e+03	180
253.1379	270	    90	        53.8000	1200	    8.6516	1.2395e+03	180
252.3950	270	    90	        53.9000	1200	    8.6113	1.2395e+03	180
251.6468	270	    90	        54	    1200	    8.5707	1.2395e+03	180
250.8932	270	    90	        54.1000	1200	    8.5298	1.2395e+03	180
250.1342	270	    90	        54.2000	1200	    8.4888	1.2395e+03	180
249.3697	270	    90	        54.3000	1200	    8.4474	1.2395e+03	180
248.5997	270	    90	        54.4000	1200	    8.4058	1.2395e+03	180
247.8239	270	    90	        54.5000	1200	    8.3640	1.2395e+03	180
247.0425	270	    90	        54.6000	1200	    8.3219	1.2395e+03	180
246.2552	270	    90	        54.7000	1200	    8.2795	1.2395e+03	180
245.4620	270	    90	        54.8000	1200	    8.2369	1.2395e+03	180
244.6629	270	    90	        54.9000	1200	    8.1940	1.2395e+03	180
243.8577	270	    90	        55	    1200	    8.1508	1.2395e+03	180
243.0463	270	    90	        55.1000	1200	    8.1073	1.2395e+03	180
242.2286	270	    90	        55.2000	1200	    8.0635	1.2395e+03	180
241.4046	270	    90	        55.3000	1200	    8.0195	1.2395e+03	180
240.5742	270	    90	        55.4000	1200	    7.9751	1.2395e+03	180
239.7372	270	    90	        55.5000	1200	    7.9305	1.2395e+03	180
238.8935	270	    90	        55.6000	1200	    7.8855	1.2395e+03	180
238.0431	270	    90	        55.7000	1200	    7.8403	1.2395e+03	180
237.1858	270	    90	        55.8000	1200	    7.7947	1.2395e+03	180
236.3215	270	    90	        55.9000	1200	    7.7488	1.2395e+03	180
235.4501	270	    90	        56	    1200	    7.7026	1.2395e+03	180
234.5714	270	    90	        56.1000	1200	    7.6560	1.2395e+03	180
233.6854	270	    90	        56.2000	1200	    7.6091	1.2395e+03	180
232.7919	270	    90	        56.3000	1200	    7.5619	1.2395e+03	180
231.8908	270	    90	        56.4000	1200	    7.5143	1.2395e+03	180
230.9820	270	    90	        56.5000	1200	    7.4663	1.2395e+03	180
230.0652	270	    90	        56.6000	1200	    7.4180	1.2395e+03	180
229.1404	270	    90	        56.7000	1200	    7.3693	1.2395e+03	180
228.2074	270	    90	        56.8000	1200	    7.3203	1.2395e+03	180
227.2661	270	    90	        56.9000	1200	    7.2708	1.2395e+03	180
226.3162	270	    90	        57	    1200	    7.2210	1.2395e+03	180
225.3576	270	    90	        57.1000	1200	    7.1707	1.2395e+03	180
224.3902	270	    90	        57.2000	1200	    7.1201	1.2395e+03	180
223.4137	270	    90	        57.3000	1200	    7.0690	1.2395e+03	180
222.4279	270	    90	        57.4000	1200	    7.0175	1.2395e+03	180
221.4328	270	    90	        57.5000	1200	    6.9656	1.2395e+03	180
220.4280	270	    90	        57.6000	1200	    6.9132	1.2395e+03	180
219.4133	270	    90	        57.7000	1200	    6.8604	1.2395e+03	180
218.3886	270	    90	        57.8000	1200	    6.8070	1.2395e+03	180
217.3536	270	    90	        57.9000	1200	    6.7533	1.2395e+03	180
216.3080	270	    90	        58	    1200	    6.6990	1.2395e+03	180
215.2517	270	    90	        58.1000	1200	    6.6442	1.2395e+03	180
214.1843	270	    90	        58.2000	1200	    6.5889	1.2395e+03	180
213.1056	270	    90	        58.3000	1200	    6.5331	1.2395e+03	180
212.0153	270	    90	        58.4000	1200	    6.4767	1.2395e+03	180
210.9131	270	    90	        58.5000	1200	    6.4198	1.2395e+03	180
209.7987	270	    90	        58.6000	1200	    6.3624	1.2395e+03	180
208.6718	270	    90	        58.7000	1200	    6.3043	1.2395e+03	180
207.5320	270	    90	        58.8000	1200	    6.2456	1.2395e+03	180
206.3790	270	    90	        58.9000	1200	    6.1863	1.2395e+03	180
205.2124	270	    90	        59	    1200	    6.1264	1.2395e+03	180
204.0319	270	    90	        59.1000	1200	    6.0659	1.2395e+03	180
202.8369	270	    90	        59.2000	1200	    6.0046	1.2395e+03	180
201.6271	270	    90	        59.3000	1200	    5.9427	1.2395e+03	180
200.4021	270	    90	        59.4000	1200	    5.8800	1.2395e+03	180
199.1612	270	    90	        59.5000	1200	    5.8167	1.2395e+03	180
197.9041	270	    90	        59.6000	1200	    5.7525	1.2395e+03	180
196.6302	270	    90	        59.7000	1200	    5.6876	1.2395e+03	180
195.3390	270	    90	        59.8000	1200	    5.6218	1.2395e+03	180
194.0297	270	    90	        59.9000	1200	    5.5552	1.2395e+03	180
192.7018	270	    90	        60.0000	1200	    5.4878	1.2395e+03	180
191.3546	270	    90	        60.1000	1200	    5.4194	1.2395e+03	180
189.9874	270	    90	        60.2000	1200	    5.3501	1.2395e+03	180
188.5994	270	    90	        60.3000	1200	    5.2798	1.2395e+03	180
187.1898	270	    90	        60.4000	1200	    5.2084	1.2395e+03	180
185.7577	270	    90	        60.5000	1200	    5.1361	1.2395e+03	180
184.3021	270	    90	        60.6000	1200	    5.0626	1.2395e+03	180
182.8220	270	    90	        60.7000	1200	    4.9880	1.2395e+03	180
181.3164	270	    90	        60.8000	1200	    4.9121	1.2395e+03	180
179.7840	270	    90	        60.9000	1200	    4.8350	1.2395e+03	180
178.2235	270	    90	        61	    1200	    4.7566	1.2395e+03	180
176.6337	270	    90	        61.1000	1200	    4.6768	1.2395e+03	180
175.0129	270	    90	        61.2000	1200	    4.5955	1.2395e+03	180
173.3594	270	    90	        61.3000	1200	    4.5127	1.2395e+03	180
171.6716	270	    90	        61.4000	1200	    4.4283	1.2395e+03	180
169.9474	270	    90	        61.5000	1200	    4.3421	1.2395e+03	180
168.1847	270	    90	        61.6000	1200	    4.2541	1.2395e+03	180
166.3809	270	    90	        61.7000	1200	    4.1642	1.2395e+03	180
164.5334	270	    90	        61.8000	1200	    4.0722	1.2395e+03	180
162.6393	270	    90	        61.9000	1200	    3.9780	1.2395e+03	180
160.6951	270	    90	        62	    1200	    3.8814	1.2395e+03	180
158.6970	270	    90	        62.1000	1200	    3.7823	1.2395e+03	180
156.6408	270	    90	        62.2000	1200	    3.6804	1.2395e+03	180
154.5214	270	    90	        62.3000	1200	    3.5755	1.2395e+03	180
152.3332	270	    90	        62.4000	1200	    3.4673	1.2395e+03	180
150.0696	270	    90	        62.5000	1200	    3.3556	1.2395e+03	180
147.7228	270	    90	        62.6000	1200	    3.2399	1.2395e+03	180
145.2836	270	    90	        62.7000	1200	    3.1198	1.2395e+03	180
142.7409	270	    90	        62.8000	1200	    2.9948	1.2395e+03	180
140.0812	270	    90	        62.9000	1200	    2.8642	1.2395e+03	180
137.2879	270	    90	        63	    1200	    2.7272	1.2395e+03	180
134.3396	270	    90	        63.1000	1200	    2.5829	1.2395e+03	180
131.2089	270	    90	        63.2000	1200	    2.4299	1.2395e+03	180
127.8589	270	    90	        63.3000	1200	    2.2664	1.2395e+03	180
124.2383	270	    90	        63.4000	1200	    2.0901	1.2395e+03	180
120.2719	270	    90	        63.5000	1200	    1.8972	1.2395e+03	180
115.8409	270	    90	        63.6000	1200	    1.6822	1.2395e+03	180
110.7377	270	    90	        63.7000	1200	    1.4351	1.2395e+03	180
104.5274	270	    90	        63.8000	1200	    1.1352	1.2395e+03	180
95.8841	    270	    90	        63.9000	1200	    0.7192	1.2395e+03	180
*)

TEST(__POUNAME());

//-----

fAngleDegrees := 8.9662;
fAngleRadians := DEG_TO_RAD(fAngleDegrees);
fExpected := 258.8987;

fResult := fbCalculateHFromAngle.CalculateH(
    Radians := fAngleRadians
);

AssertEquals_LREAL(
    Expected := fExpected,
    Actual := fResult,
    Delta := fAllowableDelta,
    Message := 'Value was not close enough to expected value.'
);

//-----

fAngleDegrees := 4.5127;
fAngleRadians := DEG_TO_RAD(fAngleDegrees);
fExpected := 173.3594;

fResult := fbCalculateHFromAngle.CalculateH(
    Radians := fAngleRadians
);

AssertEquals_LREAL(
    Expected := fExpected,
    Actual := fResult,
    Delta := fAllowableDelta,
    Message := 'Value was not close enough to expected value.'
);

//-----

fAngleDegrees := 0.7192;
fAngleRadians := DEG_TO_RAD(fAngleDegrees);
fExpected := 95.8841;

fResult := fbCalculateHFromAngle.CalculateH(
    Radians := fAngleRadians
);

AssertEquals_LREAL(
    Expected := fExpected,
    Actual := fResult,
    Delta := fAllowableDelta,
    Message := 'Value was not close enough to expected value.'
);

//-----

TEST_FINISHED();
END_METHOD

END_FUNCTION_BLOCK

// ---- Test/FB_ExternalSetpointGenerator_Test.TcPOU

FUNCTION_BLOCK FB_ExternalSetpointGenerator_Test EXTENDS FB_TestSuite
VAR
    iMotionAxis_Test1 : I_MotionAxis;
    iMotionAxis_Test2 : I_MotionAxis;

    fbExternalSetpointGenerator_Test1 : FB_ExternalSetpointGenerator(
        iMotionAxis := iMotionAxis_Test1
    );
    fbExternalSetpointGenerator_Test2 : FB_ExternalSetpointGenerator(
        iMotionAxis := iMotionAxis_Test2
    );
END_VAR


TestEnableDisableExpectEnabledDisabled_Test1();

TestSetSetpointsExpectSetpointsSet_Test2();

METHOD FB_init : BOOL
VAR_INPUT
    (* if TRUE, the retain variables are initialized (warm start / cold start)*)
    bInitRetains	: BOOL;
    (* if TRUE, the instance afterwards gets moved into the copy code (online change)*)
    bInCopyCode	: BOOL;

    MotionAxis_Test1 : I_MotionAxis;
    MotionAxis_Test2 : I_MotionAxis;
END_VAR

THIS^.iMotionAxis_Test1 := MotionAxis_Test1;
THIS^.iMotionAxis_Test2 := MotionAxis_Test2;

fbExternalSetpointGenerator_Test1.FB_Init(
    bInitRetains := FALSE,
    bInCopyCode := FALSE,
    iMotionAxis := MotionAxis_Test1
);
fbExternalSetpointGenerator_Test2.FB_Init(
    bInitRetains := FALSE,
    bInCopyCode := FALSE,
    iMotionAxis := MotionAxis_Test2
);
END_METHOD


METHOD PRIVATE TestEnableDisableExpectEnabledDisabled_Test1
VAR_INST
    nTestStep : INT;
    tonTimeout : TON;
    tTimeout : TIME := T#1s;
END_VAR

TEST(__POUNAME());

fbExternalSetpointGenerator_Test1();

CASE nTestStep OF
    0:
        IF NOT fbExternalSetpointGenerator_Test1.IsEnabled() THEN
            // Enable test can begin
            nTestStep := nTestStep + 1;
        END_IF
    1:
        IF NOT fbExternalSetpointGenerator_Test1.IsEnabled() THEN
            iMotionAxis_Test1.Power(
                Enable := TRUE,
                Enable_Positive := TRUE,
                Enable_Negative := TRUE
            );
            fbExternalSetpointGenerator_Test1.Enable();
        ELSE
            // Successfully enabled, move on
            nTestStep := nTestStep + 1;
        END_IF
    2:
        IF fbExternalSetpointGenerator_Test1.IsEnabled() THEN
            // Disable test can begin
            nTestStep := nTestStep + 1;
        END_IF
    3:
        IF fbExternalSetpointGenerator_Test1.IsEnabled() THEN
            fbExternalSetpointGenerator_Test1.Disable();
        ELSE
            // Successfully disabled, move on
            nTestStep := nTestStep + 1;
        END_IF
    4:
        // Done
END_CASE


IF nTestStep = 4 THEN
    TEST_FINISHED();
ELSIF tonTimeout.Q THEN
    AssertTrue(
        Condition := FALSE,
        Message := CONCAT('Timer timed out at step: ', TO_STRING(nTestStep))
    );

    TEST_FINISHED();
ELSE
    tonTimeout(IN := TRUE, PT := tTimeout);
END_IF
END_METHOD


METHOD PRIVATE TestSetSetpointsExpectSetpointsSet_Test2
VAR_INST
    nTestStep : INT;
    tonTimeout : TON;
    tTimeout : TIME := T#1s;

    AxisReference : REFERENCE TO AXIS_REF;
    fPositionSetpoint : LREAL := 1.0;
    fVelocitySetpoint : LREAL := 2.0;
    fAcceleraSetpoint : LREAL := 3.0;
END_VAR

TEST(__POUNAME());

fbExternalSetpointGenerator_Test2();

CASE nTestStep OF
    0:
        IF NOT fbExternalSetpointGenerator_Test2.IsEnabled() THEN
            iMotionAxis_Test2.Power(
                Enable := TRUE,
                Enable_Positive := TRUE,
                Enable_Negative := TRUE
            );
            fbExternalSetpointGenerator_Test2.Enable();
        ELSE
            // Successfully enabled, move on
            nTestStep := nTestStep + 1;
        END_IF
    1:
        IF fbExternalSetpointGenerator_Test2.IsEnabled() THEN
            // Set Setpoints test Begin

            fbExternalSetpointGenerator_Test2.SetSetpoints(
                PositionSetpoint := fPositionSetpoint,
                VelocitySetpoint := fVelocitySetpoint,
                AcceleraSetpoint := fAcceleraSetpoint,
            );

            nTestStep := nTestStep + 1;
        END_IF
    2:
        AxisReference REF= iMotionAxis_Test2.GetAxisRef();
        IF AxisReference.NcToPlc.SetVelo = fVelocitySetpoint THEN
            AssertEquals_LREAL(
                Expected := fAcceleraSetpoint,
                Actual := AxisReference.NcToPlc.SetAcc,
                Delta := 1e-3,
                Message := 'Acceleration does not have the expected setpoint.'
            );

            nTestStep := nTestStep + 1;
        END_IF
    3:
        AxisReference REF= iMotionAxis_Test2.GetAxisRef();
        IF AxisReference.NcToPlc.ActPos = fPositionSetpoint THEN
            nTestStep := nTestStep + 1;
        END_IF
    4:
        IF fbExternalSetpointGenerator_Test2.IsEnabled() THEN
            fbExternalSetpointGenerator_Test2.Disable();
        ELSE
            // Successfully disabled, move on
            nTestStep := nTestStep + 1;
        END_IF
    5:
        // Done
END_CASE


IF nTestStep = 5 THEN
    TEST_FINISHED();
ELSIF tonTimeout.Q THEN
    AssertTrue(
        Condition := FALSE,
        Message := CONCAT('Timer timed out at step: ', TO_STRING(nTestStep))
    );

    TEST_FINISHED();
ELSE
    tonTimeout(IN := TRUE, PT := tTimeout);
END_IF
END_METHOD

END_FUNCTION_BLOCK

// ---- POUs/FBs/FB_ExternalSetpointGenerator.TcPOU

FUNCTION_BLOCK FB_ExternalSetpointGenerator IMPLEMENTS I_ExternalSetpointGenerator
VAR CONSTANT
    nOFFSET_TO_NCTOPLC_AXIS_REF_STATE : DWORD := 0;
END_VAR
VAR
    iMotionAxis : I_MotionAxis;

    AxisReference : REFERENCE TO AXIS_REF;

    AxisReference_NcToPlc_StateDWord : NCTOPLC_AXIS_REF_STATE;

    bEnableCommanded : BOOL;
    fbEnableSetPointGenerator : MC_ExtSetPointGenEnable;

    bDisableCommanded : BOOL;
    fbDisableSetPointGenerator : MC_ExtSetPointGenDisable;

    bHaltCommanded : BOOL;
    fbHalt : MC_Halt;

    bEnableBusy : BOOL;
    bEnableDone : BOOL;
END_VAR


AxisReference REF= iMotionAxis.GetAxisRef();

MEMCPY(
    ADR(AxisReference_NcToPlc_StateDWord),
    ADR(AxisReference.NcToPlc) + nOFFSET_TO_NCTOPLC_AXIS_REF_STATE,
    SIZEOF(AxisReference_NcToPlc_StateDWord)
);

fbEnableSetPointGenerator(
    Axis := THIS^.AxisReference,
    Execute := bEnableCommanded
);
bEnableCommanded := FALSE;

fbDisableSetPointGenerator(
    Axis := THIS^.AxisReference,
    Execute := bDisableCommanded
);
bDisableCommanded := FALSE;

fbHalt(
    Axis := THIS^.AxisReference,
    Execute := bHaltCommanded
);
bHaltCommanded := FALSE;


METHOD PUBLIC Disable
VAR_OUTPUT
    Done : BOOL;
    Busy : BOOL;
    Error : BOOL;
    ErrorID : UDINT;
    Enabled : BOOL;
END_VAR

bDisableCommanded := TRUE;

fbDisableSetPointGenerator(
    Axis := THIS^.AxisReference,
    Done => Done,
    Busy => Busy,
    Error => Error,
    ErrorID => ErrorID,
    Enabled => Enabled
);
END_METHOD


PROPERTY DisableBusy : BOOL
GET

DisableBusy := fbDisableSetPointGenerator.Busy;
END_GET
END_PROPERTY


PROPERTY DisableDone : BOOL
GET

DisableDone := fbDisableSetPointGenerator.Done;
END_GET
END_PROPERTY


METHOD PUBLIC Enable
VAR_OUTPUT
    Done : BOOL;
    Busy : BOOL;
    Error : BOOL;
    ErrorID : UDINT;
    Enabled : BOOL;
END_VAR

IF iMotionAxis.PowerIsEnabled AND iMotionAxis.PositiveMotionIsEnabled AND iMotionAxis.NegativeMotionIsEnabled THEN
    bEnableCommanded := TRUE;
END_IF

fbEnableSetPointGenerator(
    Axis := THIS^.AxisReference,
    PositionType := E_PositionType.POSITIONTYPE_ABSOLUTE,
    Done => bEnableDone,
    Busy => bEnableBusy,
    Error => Error,
    ErrorID => ErrorID,
    Enabled => Enabled
);
END_METHOD


PROPERTY EnableBusy : BOOL
GET

EnableBusy := fbEnableSetPointGenerator.Busy;
END_GET
END_PROPERTY


PROPERTY EnableDone : BOOL
GET

EnableDone := fbEnableSetPointGenerator.Done;
END_GET
END_PROPERTY


PROPERTY EnableError : BOOL
GET

EnableError := fbEnableSetPointGenerator.Error;
END_GET
END_PROPERTY


METHOD FB_Init: BOOL
VAR_INPUT
    bInitRetains: BOOL; // TRUE: the retain variables are initialized (reset warm / reset cold)
    bInCopyCode: BOOL;  // TRUE: the instance will be copied to the copy code afterward (online change)

    iMotionAxis : I_MotionAxis;
END_VAR

THIS^.iMotionAxis := iMotionAxis;
END_METHOD


METHOD PUBLIC Halt
VAR_OUTPUT
    Done : BOOL;
    Busy : BOOL;
    Active : BOOL;
    CommandAborted : BOOL;
    Error : BOOL;
    ErrorID : UDINT;
END_VAR

fbHalt(
    Axis := THIS^.AxisReference,
    Execute := TRUE,
    Done => Done,
    Busy => Busy,
    Active => Active,
    CommandAborted => CommandAborted,
    Error => Error,
    ErrorID => ErrorID
);
END_METHOD

PROPERTY HaltBusy : BOOL
GET

HaltBusy := fbHalt.Busy;
END_GET
END_PROPERTY

PROPERTY HaltDone : BOOL
GET

HaltDone := fbHalt.Done;
END_GET
END_PROPERTY


METHOD PUBLIC IsEnabled : BOOL

IsEnabled := AxisReference_NcToPlc_StateDWord.14 AND fbEnableSetPointGenerator.Enabled;
END_METHOD


METHOD PUBLIC SetAcceleraSetpoint
VAR_INPUT
    Setpoint : LREAL;
END_VAR
VAR_OUTPUT
    Error : BOOL;
    ErrorMsg : T_MaxString;
END_VAR

SetSetpoints(
    PositionSetpoint := THIS^.AxisReference.NcToPlc.SetPos,
    VelocitySetpoint := THIS^.AxisReference.NcToPlc.SetVelo,
    AcceleraSetpoint := Setpoint,
    Error => Error,
    ErrorMsg => ErrorMsg
);
END_METHOD


METHOD PUBLIC SetPositionSetpoint
VAR_INPUT
    Setpoint : LREAL;
END_VAR
VAR_OUTPUT
    Error : BOOL;
    ErrorMsg : T_MaxString;
END_VAR

SetSetpoints(
    PositionSetpoint := Setpoint,
    VelocitySetpoint := THIS^.AxisReference.NcToPlc.SetVelo,
    AcceleraSetpoint := THIS^.AxisReference.NcToPlc.SetAcc,
    Error => Error,
    ErrorMsg => ErrorMsg
);
END_METHOD


METHOD PUBLIC SetSetpoints
VAR_INPUT
    PositionSetpoint : LREAL;
    VelocitySetpoint : LREAL;
    AcceleraSetpoint : LREAL;
END_VAR
VAR_OUTPUT
    Error : BOOL;
    ErrorMsg : T_MaxString;
END_VAR
VAR
    nDirection : DINT;
END_VAR

IF NOT THIS^.iMotionAxis.PowerIsEnabled THEN
    Error := TRUE;
    ErrorMsg := 'Cannot set external setpoint due to axis power being disabled.';
    RETURN;
END_IF

IF PositionSetpoint < THIS^.AxisReference.NcToPlc.ActPos THEN
    nDirection := -1;
ELSE
    nDirection := 1;
END_IF

IF nDirection = 1 AND NOT THIS^.iMotionAxis.PositiveMotionIsEnabled THEN
    Error := TRUE;
    ErrorMsg := 'Cannot set setpoint in the positive direction because positive motion is disabled.';
    RETURN;
END_IF

IF nDirection = -1 AND NOT THIS^.iMotionAxis.NegativeMotionIsEnabled THEN
    Error := TRUE;
    ErrorMsg := 'Cannot set setpoint in the negative direction because negative motion is disabled.';
    RETURN;
END_IF

MC_ExtSetPointGenFeed(
    Position := PositionSetpoint,
    Velocity := VelocitySetpoint,
    Acceleration := AcceleraSetpoint,
    Direction := nDirection,
    Axis := THIS^.AxisReference
);
END_METHOD


METHOD PUBLIC SetVelocitySetpoint
VAR_INPUT
    Setpoint : LREAL;
END_VAR
VAR_OUTPUT
    Error : BOOL;
    ErrorMsg : T_MaxString;
END_VAR

SetSetpoints(
    PositionSetpoint := THIS^.AxisReference.NcToPlc.SetPos,
    VelocitySetpoint := Setpoint,
    AcceleraSetpoint := THIS^.AxisReference.NcToPlc.SetAcc,
    Error => Error,
    ErrorMsg => ErrorMsg
);
END_METHOD

END_FUNCTION_BLOCK

// ---- Test/FB_HController_Test.TcPOU

FUNCTION_BLOCK FB_HController_Test EXTENDS FB_TestSuite
VAR
    MotionAxisDetAngle_Test1 : I_MotionAxis;
    MotionAxisDetH_Test1 : I_MotionAxis;
    fbCalculateHFromAngle_Test1 : FB_CalculateHFromAngle(
        D_tu := 1239.5,
        R_a := 1200,
        R_c := 90
    );
    fbExternalSetpointGenerator_Test1 : FB_ExternalSetpointGenerator(
        iMotionAxis := MotionAxisDetH_Test1
    );
    nDetAngleEncoderState1_Test1 AT %Q* : WORD;
    nDetAngleEncoderComState_Test1 AT %Q* : WORD;
END_VAR


METHOD FB_init : BOOL
VAR_INPUT
    (* if TRUE, the retain variables are initialized (warm start / cold start)*)
    bInitRetains	: BOOL;
    (* if TRUE, the instance afterwards gets moved into the copy code (online change)*)
    bInCopyCode	: BOOL;

    MotionAxisDetAngle_Test1 : I_MotionAxis;
    MotionAxisDetH_Test1 : I_MotionAxis;
END_VAR

THIS^.MotionAxisDetAngle_Test1 := MotionAxisDetAngle_Test1;
THIS^.MotionAxisDetH_Test1 := MotionAxisDetH_Test1;

fbExternalSetpointGenerator_Test1.FB_Init(
    bInitRetains := FALSE,
    bInCopyCode := FALSE,
    iMotionAxis := MotionAxisDetH_Test1
);
END_METHOD

END_FUNCTION_BLOCK
